{attribute 'GeneratedUsingTerminal: BK1250-0000-0018'}
{attribute addProperty BoxType "BK1250-0000-0018"}
{attribute addProperty Id "Term_389_KL1002KL1002_BB38DA8F0"}
{attribute addProperty CRC "2343778581"}
{attribute addProperty Size "0"}
TYPE A_0017_BK1250_0000_0018_8BB33915 EXTENDS BK1250_A2FCADE7 :
STRUCT
	{attribute addProperty Name "Term_389_KL1002"}
	Term_389_KL1002 : KL1002_BB38DA8F;
END_STRUCT
END_TYPE

(* stored: Version 1.2.0.0, ProductVersion 3.1.4024.9
   DUT A_0017_BK1250_0000_0018_8BB33915: Id {15c4fb67-2be5-4906-b03a-57a7e92d00d9} *)
